//FB sends a "command" out and waits for response of the connected device (handshake mode)
//By changing the Fnc the FB mode can be switched into only send or only receive
FUNCTION_BLOCK ComPortDeviceCom_SendRecString
VAR CONSTANT
	TIMEOUT_COM												: TIME 		:= T#10S;
END_VAR
VAR_OUTPUT CONSTANT
	FNC_SEND_REC											:	INT := 0; //Send command and wait for response
	FNC_SEND												:	INT := 1; //Send only
	FNC_REC													:	INT := 2; //Receive only
END_VAR
VAR_INPUT
	Execute													: BOOL;
	Fnc														:	INT(FNC_SEND_REC..FNC_SEND_REC) := FNC_SEND_REC;
	ClrComBuffer											: BOOL; //TRUE Clears com buffer before start
	RecTimeout												: TIME := DEFAULT_ADS_TIMEOUT; 
	Command													: T_MAxSTRing;	//Suffix will be added
	Prefix													: STRING(5) := '';
	Suffix													: STRING(5) := '$r$n';  //Will be addet to send data and removed from response
END_VAR
VAR_IN_OUT
	Handle													:	ComPortDeviceCom_BufferHandle;
END_VAR
VAR_OUTPUT
	ResponseLen												: UDINT;
	Response												: T_MaxString;
	Done													: BOOL;
	Busy													: BOOL;
	Error													: BOOL;
	ErrorID													: ComError_t := ComError_t.COMERROR_NOERROR;
END_VAR
VAR
(* Memory *****************************************************)
	state													: INT := 0;
	
(* Timer ******************************************************)
	timeout													:	ton := (PT := TIMEOUT_COM);
(* Trigger ****************************************************)
	rtExecute												: R_TRIG;
	
(* Blocks *****************************************************)
	Rec														: ReceiveString255 := (Timeout := T#10S);
	Send													: SendString255;
	
(* Error ******************************************************)
(* Dummys *****************************************************)
END_VAR

	(* Send text and receive response						 *)
	(*********************************************************)
	
(* state machine ********************************************************)
	rtExecute(CLK := Execute);
	CASE state OF
	0 : 
		Busy 												:= FALSE;
		IF NOT Execute THEN
			Done 											:= FALSE;
			Error 											:= FALSE;
			ErrorID 										:= 0;
		END_IF
		IF rtExecute.Q THEN
			Busy 											:= TRUE;		
			timeout(IN := FALSE, PT := TIMEOUT_COM + RecTimeout);
			ResponseLen 									:= 0;
			Error 											:= FALSE;
			ErrorID 										:= ComError_t.COMERROR_NOERROR;
			Rec(Reset := TRUE,Timeout := RecTimeout, rxBuffer := Handle.RxBUffer , ReceivedString := Response, Prefix := Prefix, Suffix := Suffix  );
			
			IF ClrComBuffer
			THEN
				handle.Clear();
			END_IF
			
			IF Fnc = FNC_REC
			THEN //only receive 
				MemSet(ADR(Response),0,SIZEOF(Response));
				Rec(Reset := FALSE, rxBuffer := handle.RxBUffer , ReceivedString := Response );
				State										:= 2;				
			ELSE
				Send(SendString := CONCAT(Command, Suffix),TxBuffer := Handle.TXBuffer);	
				state 										:= state + 1;
			END_IF
				
		END_IF
		
	1 : //Send tag 
		IF Send.Busy 
		THEN  //Call FB only if still busy after call in state 0
			Send(SendString := CONCAT(Command, Suffix),TxBuffer := handle.TxBuffer); 
		END_IF
		IF NOT Send.Busy 
		THEN
			IF Send.Error <> ComError_t.COMERROR_NOERROR
			THEN
				Busy										:= FALSE;
				Error										:= TRUE;
				Errorid										:= Send.Error;
				state										:= 0;
			ELSIF Fnc = FNC_SEND
			THEN
				Busy										:= FALSE;
				Done										:= TRUE;
				state										:= 0;				
			ELSE
				MemSet(ADR(Response),0,SIZEOF(Response));
				Rec(Reset := FALSE, rxBuffer := handle.RxBUffer , ReceivedString := Response );
				state 										:= state + 1;
			END_IF
		END_IF

	2: //Wair for response
		timeout(IN := TRUE);
		Rec(ReceivedString	:= Response,RXbuffer := Handle.RxBuffer);	
		IF NOT Rec.Busy
		THEN
			IF Rec.StringReceived
			THEN
				IF LEN(Response) > 0
				THEN
					IF Suffix[0] <> 0 //Cut suffix if selected 
					THEN
						Response							:= ReadStrToSeperator(Suffix,Response);
					END_IF
					ResponseLen								:= TO_UDINT(LEN(Response));	
					Busy									:= FALSE;
					Done									:= TRUE;
					state									:= 0;	
				ELSE
					; //Nothing received, continue to read until done or timeout kicks in
				END_IF
				
			ELSIF Rec.Error <> ComError_t.COMERROR_NOERROR
			THEN
				Busy										:= FALSE;
				Error										:= TRUE;
				Errorid										:= Rec.Error;
				state										:= 0;					
					
			ELSIF Rec.RxTimeout
			THEN
				Busy										:= FALSE;
				Error										:= TRUE;
				Errorid										:= ComError_t.COMERROR_TIMEOUT;
				state										:= 0;	
			ELSIF timeout.Q
			THEN
				Busy										:= FALSE;
				Error										:= TRUE;
				Errorid										:= ComError_t.COMERROR_TIMEOUT;
				state										:= 0;					
			END_IF
		END_IF
	END_CASE
(********************************************************************************)

END_FUNCTION_BLOCK

(* stored: Version 1.1.0.1, ProductVersion 3.1.4024.13
   POU ComPortDeviceCom_SendRecString: Id {7300e4f7-cfdf-4b0b-92fa-ee313b3c80fe}, SpecialFunc None *)
